{attribute 'GeneratedUsingTerminal: EL3783-0000-0018'}
{attribute addProperty BoxType "EL3783-0000-0018"}
{attribute addProperty Id "U2_SamplesAT %I*U2_Samples_1109DCAA40"}
{attribute addProperty CRC "2624712461"}
{attribute addProperty Size "40"}
TYPE L2_Voltage_Samples_9C71EF0D EXTENDS InputBase_8311D824 :
STRUCT
	{attribute addProperty Name "U2_Samples"}
	U2_Samples AT %I* : U2_Samples_1109DCAA;
END_STRUCT
END_TYPE

(* stored: Version 1.2.0.0, ProductVersion 3.1.4024.9
   DUT L2_Voltage_Samples_9C71EF0D: Id {3a6ddc3b-5b49-4d3c-a3f4-e14d44ae2c74} *)
